// TwinCAT 3 PLC project PLC1
// ProgramVersion: 3.1.4024.0
// libraries:
//   Tc2_EthernetIP, * (Beckhoff Automation GmbH)
//   Tc2_Standard, * (Beckhoff Automation GmbH)
//   Tc2_System, * (Beckhoff Automation GmbH)
//   Tc2_Utilities, * (Beckhoff Automation GmbH)
//   Tc3_Module, * (Beckhoff Automation GmbH)
// project tree:
//   DUTs/Helpers/ ST_SymAddrInfo.TcDUT
//   DUTs/ ST_CIP_COMS.TcDUT
//   GVLs/ ETHIP.TcGVL, IO.TcGVL, IP_Addresses.TcGVL
//   / PlcTask.TcTTO
//   POUs/Helpers/ FB_CIP_Client.TcPOU, FB_ReadNameByAdr.TcPOU, F_CheckIsArraySymbol.TcPOU, F_Check_Symbol_In_ETHIP.TcPOU, F_GetArrayIndexValue.TcPOU, F_ReplaceArrayIndexWithAsterisk.TcPOU, F_ScannerDevStateToString.TcPOU
//   POUs/ MAIN.TcPOU, PRG_ExtendedExample.TcPOU, PRG_SimpleExample.TcPOU, PRG_KepwareExample.TcPOU
// real-time tasks:
//   TASK PlcTask: cycle T#10ms, priority 20, ADS port 350
// I/O:
//   DEVICE Device 1 (TC3 EIP Scanner), AmsNetId 5.58.183.60.2.1
// variable links:
//   PLC1 Instance <-> Device 1 (TC3 EIP Scanner)
//     PlcTask Inputs/IO.ScannerAmsNetID <-> InfoData/AmsNetId
//     PlcTask Inputs/IO.ScannerDevState <-> Inputs/DevState

CONFIGURATION PLC1
    RESOURCE PLC ON TwinCAT3
        TASK PlcTask(INTERVAL := T#10ms, PRIORITY := 20);
        PROGRAM MAIN WITH PlcTask : MAIN;
    END_RESOURCE
END_CONFIGURATION

// ---- DUTs/Helpers/ST_SymAddrInfo.TcDUT
TYPE
    ST_SymAddrInfo :
    STRUCT
        pSymAddr : pvoid;
        cbSymSize : UDINT;
    END_STRUCT
END_TYPE

// ---- DUTs/ST_CIP_COMS.TcDUT
//Esnure that the data size, and data type name are the same on both sides.
//Was not able to make BOOL or ARRAY OF BOOL work. 
//Pack bits into other data types as needed
TYPE
    ST_CIP_COMS :
    STRUCT
        _REAL : REAL;
        _STRING : RSL5K_STRING;
        _INT : INT;
        _DINT : DINT;
        _ArrayREAL : ARRAY[0..2] OF REAL;
        _ArraySTRING : ARRAY[0..2] OF RSL5K_STRING;
        _ArrayINT : ARRAY[0..2] OF INT;
        _ArrayDINT : ARRAY[0..2] OF DINT;
    END_STRUCT
END_TYPE

// ---- GVLs/ETHIP.TcGVL
{attribute 'qualified_only'}
VAR_GLOBAL
    //"Client" variables for TwinCAT to initiate read and writes
    //Ensure there are no memory overlaps when assigning a memory address

    //Single struct example - used in "Simple Example"
    PLC1_Inputs AT %MB0 : ST_CIP_COMS; //Source of data to be written to AB from TC
    PLC1_Outputs AT %MB396 : ST_CIP_COMS; //Destination of data read from AB
	
    //Array of strucutre example used in  "Extended Example"
    arPLC_Inputs AT %MB1000 : ARRAY[0..1] OF ST_CIP_COMS; //Source of data to be written to AB from TC
    arPLC_Outputs AT %MB2000 : ARRAY[0..1] OF ST_CIP_COMS; //Destination of data read from AB	
	
	//Single Array Example - used in "Kepware Example"
    KepwareInputs : ARRAY[0..249] OF DINT; //Source of data to be written to Kepware
    KepwareOutputs :  ARRAY[0..249] OF DINT; //Destination of data read from Kepware
END_VAR

// ---- GVLs/IO.TcGVL
{attribute 'qualified_only'}
VAR_GLOBAL
    ScannerDevState AT %I* : UINT; //Linked to Device 1 (TC3 EIP Scanner)-.DevState
    ScannerAmsNetID AT %I* : AMSNETID; //Linked to Device 1 (TC3 EIP Scanner)->InfoData->AmsNetId.	    
END_VAR

// ---- GVLs/IP_Addresses.TcGVL
{attribute 'qualified_only'}
VAR_GLOBAL
	CompactLogix_1769_L16ER : STRING := '192.168.40.36';
	Kepware_Server : STRING := '192.168.40.11';
END_VAR

// ---- POUs/MAIN.TcPOU
PROGRAM MAIN
VAR
    sDevSTate : STRING;
    iSampleToRun : UINT := 0;
END_VAR

sDevSTate := F_ScannerDevStateToString(IO.ScannerDevState);

CASE iSampleToRun OF
    0:
        PRG_SimpleExample();
    1:
        PRG_ExtendedExample();
	2:
		PRG_KepwareExample();
END_CASE

END_PROGRAM

// ---- POUs/Helpers/F_ScannerDevStateToString.TcPOU
FUNCTION F_ScannerDevStateToString : STRING
VAR_INPUT
    DevState : UINT;
END_VAR
VAR
    sOut : STRING;
END_VAR

CASE DevState OF

    16#0001:
        sOut := 'Link error';
    16#0010:
        sOut := 'Out of send resources (I/O reset required)';
    16#0020:
        sOut := 'Watchdog triggered';
    16#4000:
        sOut := 'Master has no valid IP Addr - pending DHCP request';
    16#2000:
        sOut := 'TCP server: unable TO listen on local EtherNet/IP Port (44818)';
    16#1000:
        sOut := 'UDP server: unable TO listen on local EtherNet/IP Port (44818)';

END_CASE

END_FUNCTION

// ---- POUs/PRG_SimpleExample.TcPOU
PROGRAM PRG_SimpleExample
VAR
    fbRead : FB_CIP_DATA_TABLE_RDWR;
    sReadResult : STRING; //result of last read

    tonDelay : TON;
    fbWrite : FB_CIP_DATA_TABLE_RDWR;
    sWriteResult : STRING;

    iStep : UDINT;
END_VAR

CASE iStep OF

    0: //Read
        fbRead(sNetId := F_CreateAmsNetId(IO.ScannerAmsNetID), //AMS Net ID of the TwinCAT EIP Scanner 
            sIPv4Addr := IP_Addresses.CompactLogix_1769_L16ER, //IP address of the target CPU
            bExecute := TRUE,
            bDataTableWrite := FALSE, //FALSE = Read
            sSrcElementName := 'Outputs', //Name of the controller tag on the AB PLC
            sDstElementName := 'ETHIP.PLC1_Outputs', //Name of the TwinCAT variable from the "ETHIP" GVL list
            nNumberOfElements := 1, //Number of elements
            nLocalIndex := 0, //For ARRAYs the start index has to be set to indicate from which ARRAY index the data should be taken (local system)
            nRemoteIndex := 0, //For ARRAYs the start index has to be set to indicate from which ARRAY index the data should be taken (remote system)
            nSessionTimeoutMSec := 30000, //Timeout for the session
            nCmdTimeoutMSec := 7500, //Timeout for the command; 
            bRackComm := TRUE, //TRUE if the CPU is modular, i.e. a CPU with a rack design, for example a CompactLogix
            nPort := 1, //Port number of the CPU (usually 1)
            nSlot := 0, //Slot that the CPU resides in	
            bBusy =>,
            bError =>,
            nErrId =>);

        IF NOT fbRead.bBusy THEN
            fbRead(bExecute := FALSE);
            sReadResult := F_GET_ETHERNETIP_ERROR_TEXT(fbRead.nErrId);
            iStep := 10;
        END_IF

    10: //Delay timmer for simulation purposes
        tonDelay(IN := TRUE, PT := T#500MS);

        IF tonDelay.Q THEN
            tonDelay(IN := FALSE);
            iStep := 20;
        END_IF

    20: //Generate some data
        ETHIP.PLC1_Inputs._DINT := ETHIP.PLC1_Outputs._DINT + 1;
        ETHIP.PLC1_Inputs._INT := ETHIP.PLC1_Outputs._INT + 1;
        ETHIP.PLC1_Inputs._REAL := ETHIP.PLC1_Outputs._REAL + 1.1;
        ETHIP.PLC1_Inputs._STRING := STRING_TO_RSL5KSTRING(in := CONCAT('Simple Example:', TO_STRING(ETHIP.PLC1_Outputs._DINT)));
        iStep := 30;

    30: //Write
        fbWrite(sNetId := F_CreateAmsNetId(IO.ScannerAmsNetID), //AMS Net ID of the TwinCAT EIP Scanner 
            sIPv4Addr := IP_Addresses.CompactLogix_1769_L16ER, //IP address of the target CPU
            bExecute := TRUE,
            bDataTableWrite := TRUE, //TRUE = Write
            sSrcElementName := 'ETHIP.PLC1_Inputs', //Name of the TwinCAT variable from the "ETHIP" GVL list
            sDstElementName := 'Inputs', //Name of the controller tag on the AB PLC
            nNumberOfElements := 1, //Number of elements
            nLocalIndex := 0, //For ARRAYs the start index has to be set to indicate from which ARRAY index the data should be taken (local system)
            nRemoteIndex := 0, //For ARRAYs the start index has to be set to indicate from which ARRAY index the data should be taken (remote system)
            nSessionTimeoutMSec := 30000, // Timeout for the session
            nCmdTimeoutMSec := 7500, // Timeout for the command; 
            bRackComm := TRUE, //TRUE if the CPU is modular, i.e. a CPU with a rack design, for example a CompactLogix
            nPort := 1, //Port number of the CPU (usually 1)
            nSlot := 0, //Slot that the CPU resides in	
            bBusy =>,
            bError =>,
            nErrId =>);

        IF NOT fbWrite.bBusy THEN
            fbWrite(bExecute := FALSE);
            sWriteResult := F_GET_ETHERNETIP_ERROR_TEXT(fbRead.nErrId);
            iStep := 40;
        END_IF

    40: //Delay timmer for simulation purposes
        tonDelay(IN := TRUE, PT := T#500MS);

        IF tonDelay.Q THEN
            tonDelay(IN := FALSE);
            iStep := 0;
        END_IF

END_CASE

END_PROGRAM

// ---- POUs/PRG_ExtendedExample.TcPOU
//Example based on array of strucutres
PROGRAM PRG_ExtendedExample
VAR
    //An instance of FB_CIP_Client for each PLC.
    //FB_CIP_Client is just a wrapper function block of "FB_CIP_DATA_TABLE_RDWR" 
    arPLC : ARRAY[0..1] OF FB_CIP_Client;

    iStep : UDINT := 0;

    SetSourceError : BOOL;
    SetSourceErrorID : UDINT;
    SetSourceErrorTxt : STRING;

    SetReadDestError : BOOL;
    SetReadDestErrorID : UDINT;
    SetReadDestErrorTxt : STRING;

    tonIdel : TON;

    WriteError : BOOL;
    WriteErrorTxt : STRING;

    ReadError : BOOL;
    ReadErrorTxt : STRING;

    sTemp : STRING;
END_VAR


CASE iStep OF
    0: //Set the function block parameters	
        arPLC[0].NetId := F_CreateAmsNetId(IO.ScannerAmsNetID);
        arPLC[0].IPv4Addr := IP_Addresses.CompactLogix_1769_L16ER;
        arPLC[0].RackComm := TRUE;
        arPLC[0].Port := 1;
        arPLC[0].Slot := 1;
        iStep := 10;

    10: //Set the write parameters
        IF arPLC[0].SetWriteSource(pSymbol := ETHIP.arPLC_Inputs[0],
            Error => SetSourceError,
            ErrorID => SetSourceErrorID,
            ErrorTxt => SetSourceErrorTxt)
            THEN
            arPLC[0].NumberOfElementsToWrite := 1;
            arPLC[0].WriteDestination := 'Inputs';
            arPLC[0].RemoteIndexWrite := 0;

            iStep := 20;
        END_IF

    20: //Set the Read parameters
        IF arPLC[0].SetReadDest(pSymbol := ETHIP.arPLC_Outputs[0],
            Error => SetReadDestError,
            ErrorID => SetReadDestErrorID,
            ErrorTxt => SetReadDestErrorTxt)
            THEN
            arPLC[0].ReadSource := 'Outputs';
            arPLC[0].NumberOfElementsToRead := 1;
            arPLC[0].RemoteIndexRead := 0;
            iStep := 30;
        END_IF

    30: //Cycle bewteen writting and reading

        //Write
        IF arPLC[0].Write(Error => WriteError, ErrorTxt => WriteErrorTxt) THEN
            ETHIP.arPLC_Inputs[0]._DINT := ETHIP.arPLC_Outputs[0]._DINT + 1;
            ETHIP.arPLC_Inputs[0]._INT := ETHIP.arPLC_Outputs[0]._INT + 1;
            ETHIP.arPLC_Inputs[0]._REAL := ETHIP.arPLC_Outputs[0]._REAL + 1.1;
            ETHIP.arPLC_Inputs[0]._STRING := STRING_TO_RSL5KSTRING(in := CONCAT('Extended Example:', TO_STRING(ETHIP.arPLC_Outputs[0]._DINT)));
            iStep := 40;
        END_IF

    40: //Delay timmer - just for simulation
        tonIdel(IN := TRUE, PT := T#500MS);

        IF tonIdel.Q THEN
            tonIdel(IN := FALSE);
            iStep := 50;
        END_IF

    50: //Read	
        IF arPLC[0].Read(Error => ReadError, ErrorTxt => ReadErrorTxt) THEN
            iStep := 60;
            sTemp := RSL5KSTRING_TO_STRING(in := ETHIP.arPLC_Outputs[0]._STRING);
        END_IF

    60: //Delay timmer - just for simulation
        tonIdel(IN := TRUE, PT := T#500MS);

        IF tonIdel.Q THEN
            tonIdel(IN := FALSE);
            iStep := 30;
        END_IF

END_CASE

END_PROGRAM

// ---- POUs/Helpers/FB_CIP_Client.TcPOU
//Wrapper function block for "FB_CIP_DATA_TABLE_RDWR"
FUNCTION_BLOCK FB_CIP_Client
VAR
    _NetID : T_AmsNetID; //AMS Net ID of the TwinCAT EIP Scanner            			
    _IPv4Addr : STRING := '172.16.17.1'; //IP address of the target CPU
    _Slot : BYTE := 1; //Slot that the CPU resides in	
    _RackComm : BOOL := TRUE; //TRUE if the CPU is modular, i.e. a CPU with a rack design, for example a CompactLogix
    _Port : BYTE := 1; //Port number of the CPU (usually 1)

    _SessionTimeoutMSec : DWORD := 30000; // Timeout for the session
    _CmdTimeoutMSec : DWORD := 7500; // Timeout for the command; 

    //Write
    _WriteSourceSymbol : STRING(82); //Name of the variable from the "ETHIP" GVL list
    _NumberOfElementsToWrite : WORD := 1; //To write a complete UDT (structure) this should be 1
    _LocalIndexWrite : WORD := 0; //To write a complete UDT (structure) this should be 0

    _WriteDestination : STRING(82); //Name of the tag on the AB PLC
    _RemoteIndexWrite : WORD := 0; //To write a complete UDT (structure) this should be 0

    //Read
    _ReadSource : STRING(82); //Name of the tag on the AB PLC
    _NumberOfElementsToRead : WORD := 1; //To Read a complete UDT (structure) this should be 1	
    _LocalIndexRead : WORD := 0;
    _RemoteIndexRead : WORD := 0;

    _ReadDstSymbol : STRING(82); //Name of the variable from the "ETHIP" GVL List

END_VAR

;

PROPERTY CmdTimeoutMSec : DWORD
GET
CmdTimeoutMSec:=_CmdTimeoutMSec;
END_GET
SET
_CmdTimeoutMSec:=CmdTimeoutMSec;
END_SET
END_PROPERTY

//IP address of the target CPU
PROPERTY IPv4Addr : STRING
GET
IPv4Addr:=_IPv4Addr;
END_GET
SET
_IPv4Addr:=IPv4Addr;
END_SET
END_PROPERTY

//To write a complete UDT (structure) this should be 0
PROPERTY LocalIndexRead : WORD
GET
LocalIndexRead:=_LocalIndexRead;
END_GET
SET
_LocalIndexRead:=LocalIndexRead;
END_SET
END_PROPERTY

//To write a complete UDT (structure) this should be 0
PROPERTY LocalIndexWrite : WORD
GET
END_GET
SET
END_SET
END_PROPERTY

//AmsNetId of the EIP Scanner.	    
PROPERTY NetId : T_AmsNetID
GET
NetId:=_NetID;
END_GET
SET
_NetID:=NetId;
END_SET
END_PROPERTY

PROPERTY NumberOfElementsToRead : WORD
GET
NumberOfElementsToRead:=_NumberOfElementsToRead;
END_GET
SET
_NumberOfElementsToRead:=NumberOfElementsToRead;
END_SET
END_PROPERTY

//To write a complete UDT (structure) this should be 1.
PROPERTY NumberOfElementsToWrite : WORD
GET
NumberOfElementsToWrite:=_NumberOfElementsToWrite;
END_GET
SET
_NumberOfElementsToWrite:=NumberOfElementsToWrite;
END_SET
END_PROPERTY

// Port number of the CPU (usually 1)
PROPERTY Port : BYTE
GET
Port:=_Port;
END_GET
SET
_Port:=Port;
END_SET
END_PROPERTY

//TRUE if the CPU is modular, i.e. a CPU with a rack design, for example a CompactLogix
PROPERTY RackComm : BOOL
GET
RackComm:=_RackComm;
END_GET
SET
_RackComm:=RackComm;
END_SET
END_PROPERTY

METHOD Read : BOOL
VAR_INPUT
END_VAR
VAR_OUTPUT
    Error : BOOL;
    ErrId : UDINT;
    ErrorTxt : STRING;
END_VAR
VAR_INST
    GoodCnt : UDINT;
    BadCnt : UDINT;
    fbRead : FB_CIP_DATA_TABLE_RDWR;
    LastError : STRING;
    ErrorCnt : UDINT;
END_VAR
fbRead(sNetId := _NetID,
    sIPv4Addr := _IPv4Addr,
    bExecute := TRUE,
    bDataTableWrite := FALSE,
    sSrcElementName := _ReadSource,
    sDstElementName := _ReadDstSymbol,
    nNumberOfElements := _NumberOfElementsToRead,
    nLocalIndex := _LocalIndexRead,
    nRemoteIndex := _RemoteIndexRead,
    nSessionTimeoutMSec := _SessionTimeoutMSec,
    nCmdTimeoutMSec := _CmdTimeoutMSec,
    bRackComm := _RackComm,
    nPort := _Port,
    nSlot := _Slot,
    bBusy =>,
    bError => Error,
    nErrId => ErrId);

IF NOT fbRead.bBusy THEN
    IF NOT fbRead.bError THEN
        GoodCnt := GoodCnt + 1;
    ELSE
        BadCnt := BadCnt + 1;
        LastError := F_GET_ETHERNETIP_ERROR_TEXT(fbRead.nErrId);
    END_IF

    Read := TRUE;
    fbRead(bExecute := FALSE);
    ErrorTxt := F_GET_ETHERNETIP_ERROR_TEXT(fbRead.nErrId);

END_IF
END_METHOD

//Manually override the name of the variable for the destination of the read data
//Should be a variable from the "ETHIP" GVL list
PROPERTY ReadDest : STRING(82)
GET
ReadDest:=_ReadDstSymbol;
END_GET
SET
_ReadDstSymbol:=ReadDest;
END_SET
END_PROPERTY

//Name of the tag on the AB PLC
PROPERTY ReadSource : STRING
GET
ReadSource:=_ReadSource;
END_GET
SET
_ReadSource:=ReadSource;
END_SET
END_PROPERTY

PROPERTY RemoteIndexRead : WORD
GET
RemoteIndexRead:=_RemoteIndexRead;
END_GET
SET
_RemoteIndexRead:=RemoteIndexRead;
END_SET
END_PROPERTY

PROPERTY RemoteIndexWrite : WORD
GET
RemoteIndexWrite:=_RemoteIndexWrite;
END_GET
SET
_RemoteIndexWrite:=RemoteIndexWrite;
END_SET
END_PROPERTY

//Timeout for the session; the default is 30 seconds
PROPERTY SessionTimeoutMSec : DWORD
GET
SessionTimeoutMSec:=_SessionTimeoutMSec;
END_GET
SET
_SessionTimeoutMSec:=SessionTimeoutMSec;
END_SET
END_PROPERTY

//Instead of typing the name of the variable for the destination. Get the name using the variable address.
//Call untill returns true
METHOD SetReadDest : BOOL
VAR_INPUT
    pSymbol : ANY; //Variable from the ETHIP GVL list
END_VAR
VAR_OUTPUT
    Error : BOOL;
    ErrorID : UDINT;
    ErrorTxt : STRING;
END_VAR
VAR_INST
    fbGetSymbolName : FB_ReadNameByAdr;
    sTemp : STRING;
END_VAR
//Gets the name of the variable
fbGetSymbolName(pSymbol := pSymbol,
    xRead := TRUE,
    tTimeout := T#5S,
    xBusy =>,
    xError => Error,
    udiErrId => ErrorID,
    sSymName =>);

IF NOT fbGetSymbolName.xBusy THEN
    SetReadDest := TRUE;
    fbGetSymbolName(xRead := FALSE);

    IF NOT fbGetSymbolName.xError THEN
        //Check if the variable is in the "ETHIP" GVL list
        IF NOT F_Check_Symbol_In_ETHIP(sSymbolName := fbGetSymbolName.sSymName) THEN
            Error := TRUE;
            ErrorTxt := 'Variable is not declaired in the ETHIP GVL list';
            RETURN;
        END_IF

        //Check if the symbol being passed in is an array index
        IF F_CheckIsArraySymbol(sSymbolName := fbGetSymbolName.sSymName) THEN
            //Set the local read index to the array index being passed in
            _LocalIndexRead := TO_WORD(F_GetArrayIndexValue(sSymbolName := fbGetSymbolName.sSymName));
            //Replace the array index in the string with "*" 
            sTemp := F_ReplaceArrayIndexWithAsterisk(sSymbolName := fbGetSymbolName.sSymName);
        ELSE //Not an array
            sTemp := fbGetSymbolName.sSymName;
        END_IF

        //Length of the string has to be less than 82 characters
        IF LEN(sTemp) > 82 THEN
            Error := TRUE;
            ErrorTxt := CONCAT(sTemp, '| Variable name is greater than 82 characters');
            RETURN;
        END_IF

        _ReadDstSymbol := sTemp;
    END_IF
END_IF
END_METHOD

//Instead of typing the name of the variable from the "ETHIP" GVL list for the source. 
//Get the name using the variable address.
//Call untill returns true
METHOD SetWriteSource : BOOL;
VAR_INPUT
    pSymbol : ANY; //Variable from the ETHIP GVL list
END_VAR
VAR_OUTPUT
    Error : BOOL;
    ErrorID : UDINT;
    ErrorTxt : STRING;
END_VAR
VAR_INST
    fbGetSymbolName : FB_ReadNameByAdr;
    sTemp : STRING;
END_VAR
//Gets the name of the variable
fbGetSymbolName(pSymbol := pSymbol,
    xRead := TRUE,
    tTimeout := T#5S,
    xBusy =>,
    xError => Error,
    udiErrId => ErrorID,
    sSymName =>);

IF NOT fbGetSymbolName.xBusy THEN
    SetWriteSource := TRUE;
    fbGetSymbolName(xRead := FALSE);

    IF NOT fbGetSymbolName.xError THEN
        //Check if the variable is in the "ETHIP" GVL list
        IF NOT F_Check_Symbol_In_ETHIP(sSymbolName := fbGetSymbolName.sSymName) THEN
            Error := TRUE;
            ErrorTxt := 'Variable is not declaired in the ETHIP GVL list';
            RETURN;
        END_IF

        //Check if the symbol being passed in is an array index
        IF F_CheckIsArraySymbol(sSymbolName := fbGetSymbolName.sSymName) THEN
            //Set the local write index to the array index being passed in
            _LocalIndexWrite := TO_WORD(F_GetArrayIndexValue(sSymbolName := fbGetSymbolName.sSymName));
            //Replace the 
            sTemp := F_ReplaceArrayIndexWithAsterisk(sSymbolName := fbGetSymbolName.sSymName);
        ELSE //Not an array
            sTemp := fbGetSymbolName.sSymName;
        END_IF

        //Length of the string has to be less than 82 characters
        IF LEN(sTemp) > 82 THEN
            Error := TRUE;
            ErrorTxt := CONCAT(sTemp, '| Variable name is greater than 82 characters');
            RETURN;
        END_IF

        _WriteSourceSymbol := sTemp;

    END_IF

END_IF
END_METHOD

//Slot number if the CPU is not plugged into slot 0
PROPERTY Slot : BYTE
GET
Slot:=_Slot;
END_GET
SET
_Slot:=Slot;
END_SET
END_PROPERTY

//Write Data to the target, call untill returns true
METHOD PUBLIC Write : BOOL
VAR_INPUT
END_VAR
VAR_OUTPUT
    Error : BOOL;
    ErrId : UDINT;
    ErrorTxt : STRING;
END_VAR
VAR_INST
    GoodCnt : UDINT;
    BadCnt : UDINT;
    fbWrite : FB_CIP_DATA_TABLE_RDWR;
    LastError : STRING;
    ErrorCnt : UDINT;
END_VAR
fbWrite(sNetId := _NetID,
    sIPv4Addr := _IPv4Addr,
    bExecute := TRUE,
    bDataTableWrite := TRUE,
    sSrcElementName := _WriteSourceSymbol,
    sDstElementName := _WriteDestination,
    nNumberOfElements := _NumberOfElementsToWrite,
    nLocalIndex := _LocalIndexWrite,
    nRemoteIndex := _RemoteIndexWrite,
    nSessionTimeoutMSec := _SessionTimeoutMSec,
    nCmdTimeoutMSec := _CmdTimeoutMSec,
    bRackComm := _RackComm,
    nPort := _Port,
    nSlot := _Slot,
    bBusy =>,
    bError => Error,
    nErrId => ErrId);

IF NOT fbWrite.bBusy THEN
    IF NOT fbWrite.bError THEN
        GoodCnt := GoodCnt + 1;
    ELSE
        BadCnt := BadCnt + 1;
        LastError := F_GET_ETHERNETIP_ERROR_TEXT(fbWrite.nErrId);
    END_IF

    Write := TRUE;
    fbWrite(bExecute := FALSE);
    ErrorTxt := F_GET_ETHERNETIP_ERROR_TEXT(fbWrite.nErrId);
END_IF
END_METHOD

//Name of the controller tag on the AB PLC
PROPERTY WriteDestination : STRING(82)
GET
WriteDestination:=_WriteDestination;
END_GET
SET
_WriteDestination:=WriteDestination;
END_SET
END_PROPERTY

//Manually override the name of the source variable to be written
//Should be a variable from the "ETHIP" GVL list
PROPERTY WriteSource : STRING(82)
GET
WriteSource:=_WriteSourceSymbol;
END_GET
SET
_WriteSourceSymbol:=WriteSource;
END_SET
END_PROPERTY

END_FUNCTION_BLOCK

// ---- POUs/Helpers/FB_ReadNameByAdr.TcPOU
FUNCTION_BLOCK FB_ReadNameByAdr
VAR_INPUT
    pSymbol : ANY;
    xRead : BOOL;
    tTimeout : TIME := T#5S;
END_VAR
VAR_OUTPUT
    xBusy : BOOL;
    xError : BOOL;
    udiErrId : UDINT;
    sSymName : T_MaxString;
END_VAR
VAR
    fbAdsRWEx : ADSRDWRTEX;
    stADRInfo : ST_SymAddrInfo;
    fbRT : R_TRIG;
END_VAR

fbRT(CLK := xRead);

IF fbRT.Q THEN
    xBusy := TRUE;
    xError := FALSE;
    udiErrId := 0;

    stADRInfo.pSymAddr := pSymbol.pValue;
    stADRInfo.cbSymSize := TO_UDINT(pSymbol.diSize);
    MEMSET(ADR(sSymName), 0, SIZEOF(sSymName));

    fbAdsRWEx(WRTRD := FALSE);
    fbAdsRWEx(NETID := '',
        PORT := _AppInfo.AdsPort,
        IDXGRP := 16#40A1,
        IDXOFFS := 0,
        DESTADDR := ADR(sSymName),
        READLEN := SIZEOF(sSymName),
        SRCADDR := ADR(stADRInfo),
        WRITELEN := SIZEOF(stADRInfo),
        WRTRD := TRUE,
        TMOUT := tTimeout);
ELSE
    fbAdsRWEx(WRTRD := FALSE, BUSY => xBusy, ERR => xError, ERRID => udiErrID);
END_IF

END_FUNCTION_BLOCK

// ---- POUs/Helpers/F_Check_Symbol_In_ETHIP.TcPOU
//returns true if part of the "ETHIP" GVL List.
FUNCTION F_Check_Symbol_In_ETHIP : BOOL
VAR_INPUT
    sSymbolName : STRING;
END_VAR
VAR
END_VAR

IF LEFT(sSymbolName, 6) = 'ETHIP.' THEN
    F_Check_Symbol_In_ETHIP := TRUE;
ELSE
    F_Check_Symbol_In_ETHIP := FALSE;
END_IF

END_FUNCTION

// ---- POUs/Helpers/F_CheckIsArraySymbol.TcPOU
//Check if the symbol string is an array, i.e. contains "[ ]"
FUNCTION F_CheckIsArraySymbol : BOOL
VAR_INPUT
    sSymbolName : STRING;
END_VAR
VAR
    iOpenBrackLocation : INT;
    iClosedBracketLocation : INT;
END_VAR

iOpenBrackLocation := FIND(sSymbolName, '[');
iClosedBracketLocation := FIND(sSymbolName, ']');

IF iOpenBrackLocation <> 0 AND iClosedBracketLocation > iOpenBrackLocation THEN
    F_CheckIsArraySymbol := TRUE;

ELSE
    F_CheckIsArraySymbol := FALSE;
END_IF

END_FUNCTION

// ---- POUs/Helpers/F_GetArrayIndexValue.TcPOU
//Given a symbol string like "ETHIP.arData[10]".
//Return the value bewteen "[]" i.e. 10.
FUNCTION F_GetArrayIndexValue : DINT
VAR_INPUT
    sSymbolName : STRING;
END_VAR
VAR
    iOpenBrackLocation : INT;
    iClosedBracketLocation : INT;
    iNumOfCharsInIndex : INT;
    sIndex : STRING;
END_VAR

iOpenBrackLocation := FIND(sSymbolName, '[');
iClosedBracketLocation := FIND(sSymbolName, ']');

IF iOpenBrackLocation <> 0 AND iClosedBracketLocation > iOpenBrackLocation THEN
    iNumOfCharsInIndex := (iClosedBracketLocation - iOpenBrackLocation) - 1;

    sIndex := MID(STR := sSymbolName, LEN := iNumOfCharsInIndex, POS := iOpenBrackLocation + 1);

    F_GetArrayIndexValue := TO_DINT(sIndex);
END_IF

END_FUNCTION

// ---- POUs/Helpers/F_ReplaceArrayIndexWithAsterisk.TcPOU
FUNCTION F_ReplaceArrayIndexWithAsterisk : STRING
VAR_INPUT
    sSymbolName : STRING;
END_VAR
VAR
    iOpenBrackLocation : INT;
    iClosedBracketLocation : INT;
    iNumOfCharsInIndex : INT;
END_VAR

iOpenBrackLocation := FIND(sSymbolName, '[');
iClosedBracketLocation := FIND(sSymbolName, ']');

IF iOpenBrackLocation <> 0 AND iClosedBracketLocation > iOpenBrackLocation THEN
    iNumOfCharsInIndex := (iClosedBracketLocation - iOpenBrackLocation) - 1;
    F_ReplaceArrayIndexWithAsterisk := REPLACE(STR1 := sSymbolName, STR2 := '*', L := iNumOfCharsInIndex, P := iOpenBrackLocation + 1);
ELSE
    F_ReplaceArrayIndexWithAsterisk := sSymbolName;
END_IF

END_FUNCTION

// ---- POUs/PRG_KepwareExample.TcPOU
PROGRAM PRG_KepwareExample
VAR
    fbRead : FB_CIP_DATA_TABLE_RDWR;
    sReadResult : STRING; //result of last read

    tonDelay : TON;
    fbWrite : FB_CIP_DATA_TABLE_RDWR;
    sWriteResult : STRING;

    iStep : UDINT;
END_VAR

CASE iStep OF

    0: //Read
        fbRead(sNetId := F_CreateAmsNetId(IO.ScannerAmsNetID), //AMS Net ID of the TwinCAT EIP Scanner 
            sIPv4Addr := IP_Addresses.Kepware_Server, //IP address of the target CPU
            bExecute := TRUE,
            bDataTableWrite := FALSE, //FALSE = Read
            sSrcElementName := 'Outputs.HostComData[0]', //Name of the controller tag on the Kepware
            sDstElementName := 'ETHIP.KepwareOutputs[0]', //Name of the TwinCAT variable from the "ETHIP" GVL list
            nNumberOfElements := 250, //Number of elements
            nLocalIndex := 0, //For ARRAYs the start index has to be set to indicate from which ARRAY index the data should be taken (local system)
            nRemoteIndex := 0, //For ARRAYs the start index has to be set to indicate from which ARRAY index the data should be taken (remote system)
            nSessionTimeoutMSec := 30000, //Timeout for the session
            nCmdTimeoutMSec := 7500, //Timeout for the command; 
            bRackComm := FALSE, //TRUE if the CPU is modular, i.e. a CPU with a rack design, for example a CompactLogix
            nPort := 1, //Port number of the CPU (usually 1)
            nSlot := 1, //Slot that the CPU resides in	
            bBusy =>,
            bError =>,
            nErrId =>);

        IF NOT fbRead.bBusy THEN
            fbRead(bExecute := FALSE);
            sReadResult := F_GET_ETHERNETIP_ERROR_TEXT(fbRead.nErrId);
            iStep := 10;
        END_IF

    10: //Delay timmer for simulation purposes
        tonDelay(IN := TRUE, PT := T#500MS);

        IF tonDelay.Q THEN
            tonDelay(IN := FALSE);
            iStep := 20;
        END_IF

    20: //Generate some data
        ETHIP.PLC1_Inputs._DINT := ETHIP.PLC1_Outputs._DINT + 1;
        ETHIP.PLC1_Inputs._INT := ETHIP.PLC1_Outputs._INT + 1;
        ETHIP.PLC1_Inputs._REAL := ETHIP.PLC1_Outputs._REAL + 1.1;
        ETHIP.PLC1_Inputs._STRING := STRING_TO_RSL5KSTRING(in := CONCAT('Simple Example:', TO_STRING(ETHIP.PLC1_Outputs._DINT)));
        iStep := 30;

    30: //Write
        fbWrite(sNetId := F_CreateAmsNetId(IO.ScannerAmsNetID), //AMS Net ID of the TwinCAT EIP Scanner 
            sIPv4Addr := IP_Addresses.Kepware_Server, //IP address of the target CPU
            bExecute := TRUE,
            bDataTableWrite := TRUE, //TRUE = Write
            sSrcElementName := 'ETHIP.KepwareInputs[0]', //Name of the TwinCAT variable from the "ETHIP" GVL list
            sDstElementName := 'Inputs.HostComData[0]', //Name of the controller tag on the Kepware
            nNumberOfElements := 250, //Number of elements
            nLocalIndex := 0, //For ARRAYs the start index has to be set to indicate from which ARRAY index the data should be taken (local system)
            nRemoteIndex := 0, //For ARRAYs the start index has to be set to indicate from which ARRAY index the data should be taken (remote system)
            nSessionTimeoutMSec := 30000, // Timeout for the session
            nCmdTimeoutMSec := 7500, // Timeout for the command; 
            bRackComm := FALSE, //TRUE if the CPU is modular, i.e. a CPU with a rack design, for example a CompactLogix
            nPort := 1, //Port number of the CPU (usually 1)
            nSlot := 1, //Slot that the CPU resides in	
            bBusy =>,
            bError =>,
            nErrId =>);

        IF NOT fbWrite.bBusy THEN
            fbWrite(bExecute := FALSE);
            sWriteResult := F_GET_ETHERNETIP_ERROR_TEXT(fbRead.nErrId);
            iStep := 40;
        END_IF

    40: //Delay timmer for simulation purposes
        tonDelay(IN := TRUE, PT := T#500MS);

        IF tonDelay.Q THEN
            tonDelay(IN := FALSE);
            iStep := 0;
        END_IF

END_CASE

END_PROGRAM
